// TIA Portal V20 export
VAR_GLOBAL   // PLC tag table "Unit1Em4"
   "BA010AZCRPM04.04" AT %Q2012.4 : Bool;   // FEEDER CYLINDER DOWN
   "BA010AZCRPM04.05" AT %Q2012.5 : Bool;   // FEEDER CYLINDER UP
   "BA010AZCRBK05.04" AT %I1016.4 : Bool;   // FEEDER CYLINDER UP
   "BA010AZCRBK05.13" AT %I1017.3 : Bool;   // COMPENSATOR SAFETY PIN IDLE POSITION
   "BA010AZCRBK05.14" AT %I1017.4 : Bool;   // FEEDER CYLINDER DOWN
   "BA010AZCRSP503.03" AT %IW3106 : Int;   // CUTTER EPC SENSOR
END_VAR
VAR_GLOBAL CONSTANT   // user constants
   U1EM4_NO_OF_AXES : USInt := 5;   // Starts with 1. E.g., the value 4 means that 4 axes exist.
   DR3_RatedTorque : LReal := 1.27;   // CompensatorAxisZ
   DR4_RatedTorque : LReal := 1.27;   // FeedingRollAxisB
   DR5_RatedTorque : LReal := 1.27;   // ElectordCutterAxisZ
   DR6_RatedTorque : LReal := 1.27;   // PositionMovingAxisX
   U1EM4_JOB01 : DInt := 1;
   U1EM4_JOB02 : DInt := 2;
   U1EM4_JOB03 : DInt := 3;
   U1EM4_JOB04 : DInt := 4;
   U1EM4_JOB05 : DInt := 5;
   U1EM4_JOB06 : DInt := 6;
   U1EM4_JOB07 : DInt := 7;
   U1EM4_JOB08 : DInt := 8;
   U1EM4_JOB09 : DInt := 9;
   U1EM4_JOB10 : DInt := 10;
   U1EM4_JOB11 : DInt := 11;
   U1EM4_JOB12 : DInt := 12;
   U1EM4_JOB13 : DInt := 13;
   U1EM4_JOB14 : DInt := 14;
   U1EM4_JOB15 : DInt := 15;
   U1EM4_JOB16 : DInt := 16;
   U1EM4_JOB17 : DInt := 17;
   U1EM4_JOB18 : DInt := 18;
   U1EM4_JOB19 : DInt := 19;
   U1EM4_JOB20 : DInt := 20;
   U1EM4_JOB21 : DInt := 21;
   U1EM4_JOB22 : DInt := 22;
   U1EM4_JOB23 : DInt := 23;
   U1EM4_JOB24 : DInt := 24;
   U1EM4_JOB25 : DInt := 25;
   U1EM4_JOB26 : DInt := 26;
   U1EM4_JOB27 : DInt := 27;
   U1EM4_JOB28 : DInt := 28;
   U1EM4_JOB29 : DInt := 29;
   U1EM4_JOB30 : DInt := 30;
   U1EM4_JOB31 : DInt := 31;
   U1EM4_JOB32 : DInt := 32;
   U1EM4_JOB33 : DInt := 33;
   U1EM4_JOB34 : DInt := 34;
   U1EM4_JOB35 : DInt := 35;
   U1EM4_JOB36 : DInt := 36;
   U1EM4_JOB37 : DInt := 37;
   U1EM4_JOB38 : DInt := 38;
   U1EM4_JOB39 : DInt := 39;
   U1EM4_JOB40 : DInt := 40;
   U1EM4_JOB41 : DInt := 41;
   U1EM4_JOB42 : DInt := 42;
   U1EM4_JOB43 : DInt := 43;
   U1EM4_JOB44 : DInt := 44;
   U1EM4_JOB45 : DInt := 45;
   U1EM4_JOB46 : DInt := 46;
   U1EM4_JOB47 : DInt := 47;
   U1EM4_JOB48 : DInt := 48;
   U1EM4_JOB49 : DInt := 49;
   U1EM4_JOB50 : DInt := 50;
END_VAR
